# EPICS autosave request: iocBoot/iocmmc100/auto_settings.req
file motor_settings.req P=MLL:,M=sphi
